(* PLC project Tc3_EventLogger.GetAlarmEx Demo, tc3-libraries-kb TwinCAT 3.1 *)
(* stored: creationDateTime 2026-05-11T01:00:00, modificationDateTime 2026-05-11T01:00:00 *)

PROGRAM P_Demo_GetAlarmEx
  VAR
    fbGetAlarmEx : GetAlarmEx;  (* Tc3_EventLogger.GetAlarmEx 实例 *)
    arg_stEventEntry : TcEventEntry;  (* VAR_INPUT stEventEntry *)
    arg_ipSourceInfo : I_TcSourceInfo;  (* VAR_INPUT ipSourceInfo *)
    arg_fbAlarm : REFERENCE TO FB_TcAlarm;  (* VAR_INPUT fbAlarm *)
  END_VAR

            // ============================================================
// Tc3_EventLogger.GetAlarmEx 演示程序（FB 实例）
// ============================================================
// 验证步骤：
//   1. 引用 Tc3_EventLogger（及依赖类型所在库 Tc2_System 等）
//   2. 编译 + 登录
//   3. 按 doc.md 给 arg_* 赋值
//   4. 在线监视 out_* / io_* 输出
// ============================================================

fbGetAlarmEx(
    stEventEntry := arg_stEventEntry,
    ipSourceInfo := arg_ipSourceInfo,
    fbAlarm := arg_fbAlarm
);

          
END_PROGRAM
